// TIA Portal project "hmi_deneme" (V18)

(* hardware
DEVICE "HMI_1"  TP700 Comfort
   slot 0: "HMI_1"  TP700 Comfort  6AV2 124-0GC01-0AX0  17.0.0.0
   slot 1: "HMI_RT_1"  TP700 Comfort  6AV2 124-0GC01-0AX0  17.0.0.0
   slot 5: "HMI_1.IE_CP_1"  PROFINET Interface  17.0.0.0
      slot 1: "PROFINET Interface_1"  PROFINET Interface
         slot 1: "Port_1"  Port
         slot 2: "Port_2"  Port
   slot 7: "HMI_1.MPI/DP_CP_1"  MPI/DP Interface  17.0.0.0
DEVICE "S7-1200 station_1"  S7-1200 Station
   slot 0: "Rack_0"  S7-1200 Rack  Rack  V1.0
   slot 1: "PLC_1"  CPU 1215C DC/DC/DC  6ES7 215-1AG40-0XB0  V4.5
*)

// ===== PLC "PLC_1"  CPU 1215C DC/DC/DC =====

VAR_GLOBAL   // PLC tag table "Default tag table"
   "B0" AT %M0.0 : Bool;
   "B1" AT %M0.1 : Bool;
   "B2" AT %M0.2 : Bool;
   "B3" AT %M0.3 : Bool;
   "BTN" AT %I0.0 : Bool;
   "M0" AT %M1.0 : Bool;
   "A1" AT %M2.0 : Bool;
   "A2" AT %M2.1 : Bool;
   "M1" AT %M1.1 : Bool;
   "A3" AT %M2.2 : Bool;
   "M2" AT %M1.2 : Bool;
   "L1" AT %Q0.0 : Bool;
   "L2" AT %Q0.1 : Bool;
   "L3" AT %Q0.2 : Bool;
   "L4" AT %Q0.3 : Bool;
END_VAR

FUNCTION "Block_1" : Void   // FC1, LAD
{ S7_Optimized_Access := 'TRUE' }
VERSION : 0.1
   VAR_TEMP   // added for the SCL form of the ladder/FBD networks
      _w1 : Bool;
   END_VAR
BEGIN

REGION Network 1
   // BIT0
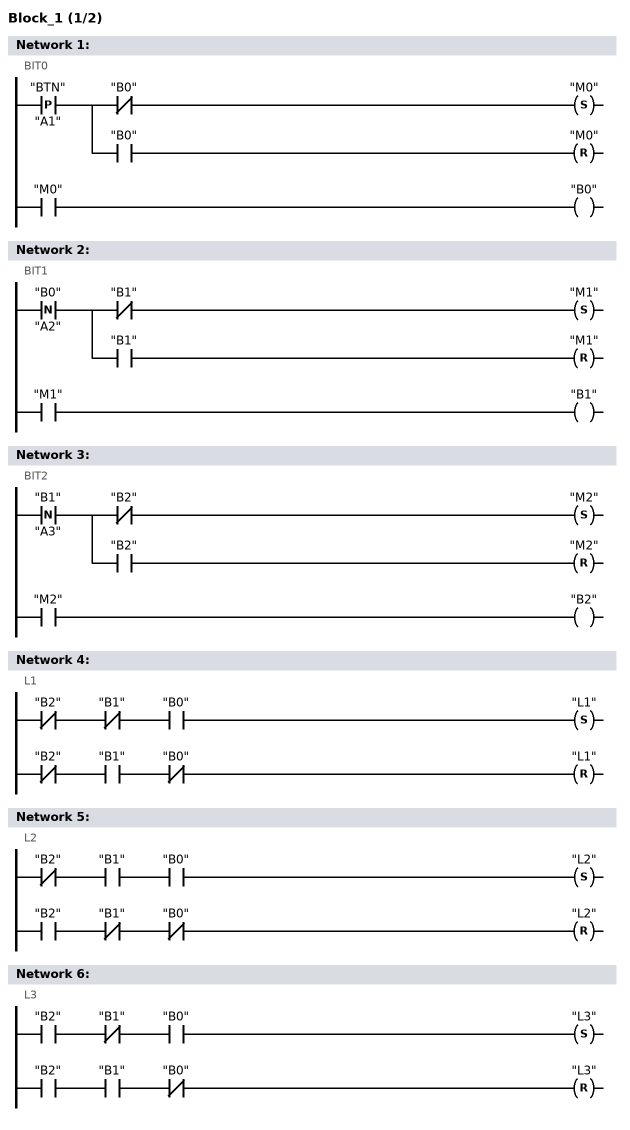
   RUNG wire#powerrail
      P_Contact(operand := "BTN", bit := "A1")
      wire#w1
      I_Contact( "B0" )
      S_Coil( "M0" )
   END_RUNG
   RUNG wire#w1
      Contact( "B0" )
      R_Coil( "M0" )
   END_RUNG
   RUNG wire#powerrail
      Contact( "M0" )
      Coil( "B0" )
   END_RUNG
   // the same network as SCL:
   #_w1 := "BTN" AND NOT "A1";   // rising edge of "BTN"
   "A1" := "BTN";
   IF #_w1 AND NOT "B0" THEN "M0" := TRUE; END_IF;
   IF #_w1 AND "B0" THEN "M0" := FALSE; END_IF;
   "B0" := "M0";
END_REGION

REGION Network 2
   // BIT1
   RUNG wire#powerrail
      N_Contact(operand := "B0", bit := "A2")
      wire#w1
      I_Contact( "B1" )
      S_Coil( "M1" )
   END_RUNG
   RUNG wire#w1
      Contact( "B1" )
      R_Coil( "M1" )
   END_RUNG
   RUNG wire#powerrail
      Contact( "M1" )
      Coil( "B1" )
   END_RUNG
   // the same network as SCL:
   #_w1 := NOT "B0" AND "A2";   // falling edge of "B0"
   "A2" := "B0";
   IF #_w1 AND NOT "B1" THEN "M1" := TRUE; END_IF;
   IF #_w1 AND "B1" THEN "M1" := FALSE; END_IF;
   "B1" := "M1";
END_REGION

REGION Network 3
   // BIT2
   RUNG wire#powerrail
      N_Contact(operand := "B1", bit := "A3")
      wire#w1
      I_Contact( "B2" )
      S_Coil( "M2" )
   END_RUNG
   RUNG wire#w1
      Contact( "B2" )
      R_Coil( "M2" )
   END_RUNG
   RUNG wire#powerrail
      Contact( "M2" )
      Coil( "B2" )
   END_RUNG
   // the same network as SCL:
   #_w1 := NOT "B1" AND "A3";   // falling edge of "B1"
   "A3" := "B1";
   IF #_w1 AND NOT "B2" THEN "M2" := TRUE; END_IF;
   IF #_w1 AND "B2" THEN "M2" := FALSE; END_IF;
   "B2" := "M2";
END_REGION

REGION Network 4
   // L1
   RUNG wire#powerrail
      I_Contact( "B2" )
      I_Contact( "B1" )
      Contact( "B0" )
      S_Coil( "L1" )
   END_RUNG
   RUNG wire#powerrail
      I_Contact( "B2" )
      Contact( "B1" )
      I_Contact( "B0" )
      R_Coil( "L1" )
   END_RUNG
   // the same network as SCL:
   IF NOT "B2" AND NOT "B1" AND "B0" THEN "L1" := TRUE; END_IF;
   IF NOT "B2" AND "B1" AND NOT "B0" THEN "L1" := FALSE; END_IF;
END_REGION

REGION Network 5
   // L2
   RUNG wire#powerrail
      I_Contact( "B2" )
      Contact( "B1" )
      Contact( "B0" )
      S_Coil( "L2" )
   END_RUNG
   RUNG wire#powerrail
      Contact( "B2" )
      I_Contact( "B1" )
      I_Contact( "B0" )
      R_Coil( "L2" )
   END_RUNG
   // the same network as SCL:
   IF NOT "B2" AND "B1" AND "B0" THEN "L2" := TRUE; END_IF;
   IF "B2" AND NOT "B1" AND NOT "B0" THEN "L2" := FALSE; END_IF;
END_REGION

REGION Network 6
   // L3
   RUNG wire#powerrail
      Contact( "B2" )
      I_Contact( "B1" )
      Contact( "B0" )
      S_Coil( "L3" )
   END_RUNG
   RUNG wire#powerrail
      Contact( "B2" )
      Contact( "B1" )
      I_Contact( "B0" )
      R_Coil( "L3" )
   END_RUNG
   // the same network as SCL:
   IF "B2" AND NOT "B1" AND "B0" THEN "L3" := TRUE; END_IF;
   IF "B2" AND "B1" AND NOT "B0" THEN "L3" := FALSE; END_IF;
END_REGION

REGION Network 7
   // L4
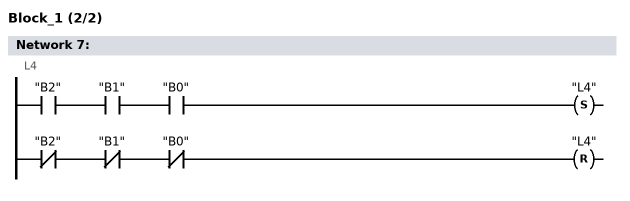
   RUNG wire#powerrail
      Contact( "B2" )
      Contact( "B1" )
      Contact( "B0" )
      S_Coil( "L4" )
   END_RUNG
   RUNG wire#powerrail
      I_Contact( "B2" )
      I_Contact( "B1" )
      I_Contact( "B0" )
      R_Coil( "L4" )
   END_RUNG
   // the same network as SCL:
   IF "B2" AND "B1" AND "B0" THEN "L4" := TRUE; END_IF;
   IF NOT "B2" AND NOT "B1" AND NOT "B0" THEN "L4" := FALSE; END_IF;
END_REGION
END_FUNCTION

ORGANIZATION_BLOCK "Main"   // OB1, LAD, ProgramCycle
TITLE = "Main Program Sweep (Cycle)"
{ S7_Optimized_Access := 'TRUE' }
VERSION : 0.1
   VAR_INPUT
      Initial_Call : Bool;   // Initial call of this OB
      Remanence : Bool;   // =True, if remanent data are available
   END_VAR
BEGIN

REGION Network 1
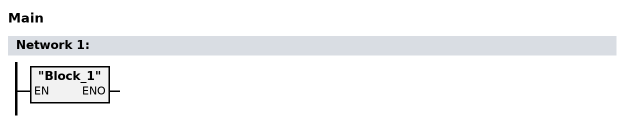
   RUNG wire#powerrail
      "Block_1"()
   END_RUNG
   // the same network as SCL:
   "Block_1"();
END_REGION
END_ORGANIZATION_BLOCK

(* ===== HMI "HMI_RT_1" =====
system functions are stored by id; their names below are inferred from use
connection "HMI_Connection_1": ETHERNET, S7_1200_OMS

HMI tags "Default tag table"
   "HMI" : Bool = PLC BTN AT %I0.0, 1 s

HMI tags "DEmo Tags"
   "Bit_1" : Bool, internal
   "Bit_2" : Bool, internal
   "Word_1" : Int, internal
   "Word_2" : Int, internal
   "AlarmTriggerWord" : UInt, internal
   "CurrentUserName" : WString[254], internal
   "CurrentGroup" : Int, internal

discrete alarms
   4: 'Warning 2', class Warnings, trigger "AlarmTriggerWord" bit 3
   3: 'Warning 1', class Warnings, trigger "AlarmTriggerWord" bit 2
   2: 'Alarm 2', class Errors, trigger "AlarmTriggerWord" bit 1
   1: 'Alarm 1', class Errors, trigger "AlarmTriggerWord" bit 0

text list "OFF_ON_List": 0 'OFF'; 1 'ON'

recipe "Recipe_1": Recipe_element_1 <- "Word_1", Recipe_element_2 <- "Word_2"

SlideinScreen "GraphX_Slidein_Left" 270x480
   TextField "Text field_1" at 28,20 size 224x23; Text 'Slide in from left screen'
   Button "Button_1" at 16,433 size 239x32; TextOff 'Close'
      on Press: function_cf6f4242("GraphX_Slidein_Left", 0)

Template "ScrNav" 800x430
   Button "Template_Button_1" at 6,391 size 192x32; TextOff 'Home'
      on Click: ActivateScreen("Home", 0)
   Button "Template_Button_2" at 205,391 size 192x32; TextOff 'Toolbox'
      on Click: ActivateScreen("Toolbox", 0)
   Button "Template_Button_3" at 404,391 size 192x32; TextOff 'Alarms'
      on Click: ActivateScreen("Alarms", 0)
   Button "Template_Button_4" at 602,391 size 192x32; TextOff 'Trend'
      on Click: ActivateScreen("Trend", 0)
   Button "Template_Button_5" at 6,353 size 192x32; TextOff 'Recipe'
      on Click: ActivateScreen("Recipe", 0)
   Button "Template_Button_6" at 205,353 size 192x32; TextOff 'UserAdmin'
      on Click: ActivateScreen("UserAdmin", 0)

screen "Home" 800x430, template "ScrNav"
   TextField "Text field_1" at 638,22 size 123x23; Text 'Home Screen'
   Button "Button_1" at 26,26 size 192x32; TextOff 'Help Popup'
      on Click: function_efd93a16("Help Popup", 0, 0, -1, -1, 1)
   Button "Button_2" at 26,73 size 192x32; TextOn 'Help Popup'; TextOff 'Show Slide in Left'
      on Press: function_cf6f4242("GraphX_Slidein_Left", 1)

screen "Toolbox" 800x430, template "ScrNav"
   TextField "Text field_1" at 629,22 size 145x23; Text 'Toolbox Screen'
   Button "Button_1" at 42,32 size 186x89; TextOff 'Momentary'; TextList "OFF_ON_List"
      on Press: function_b14e0dd5("Bit_1", 0)
      Appearance <- "Bit_1"
      ProcessValue <- "Bit_1"
   IOField "I/O field_1" at 273,32 size 93x89; FormatPattern 1
      ProcessValue <- "Bit_1"
   Circle "Circle_1" at 402,49 size 48x48
      Visibility <- "Bit_1"
   SymbolicIOField "Symbolic I/O field_1" at 480,50 size 112x46; TextOff '0'; TextOn '1'; TextList "OFF_ON_List"
      ProcessValue <- "Bit_1"

PopupScreen "Help Popup" 240x240
   Button "Button_1" at 18,198 size 197x31; TextOff 'Close'
      on Press: function_efd93a16("Help Popup", 0, 0, 0, -1, 1)
   TextField "Text field_1" at 61,34 size 108x23; Text 'Help Popup'

screen "Trend" 800x430, template "ScrNav"
   IOField "I/O field_1" at 135,14 size 96x32; FormatPattern s99999
      ProcessValue <- "Word_1"
   IOField "I/O field_2" at 395,16 size 96x32; FormatPattern s99999
      ProcessValue <- "Word_2"
   TextField "Text field_1" at 53,19 size 74x23; Text 'Word_1'
   TextField "Text field_2" at 311,19 size 74x23; Text 'Word_2'
   TrendView "Trend view_1" at 20,62 size 762x312

screen "Alarms" 800x430, template "ScrNav"
   TextField "Text field_1" at 47,38 size 226x23; Text 'Alarm Trigger Word Bits'
   IOField "I/O field_1" at 281,33 size 96x32; FormatPattern 1111
      ProcessValue <- "AlarmTriggerWord"
   AlarmView "Alarm view_1" at 49,73 size 715x165
   AlarmView "Alarm view_2" at 49,241 size 716x139

screen "Recipe" 800x430, template "ScrNav"
   IOField "I/O field_1" at 135,14 size 96x32; FormatPattern s99999
      ProcessValue <- "Word_1"
   IOField "I/O field_2" at 395,16 size 96x32; FormatPattern s99999
      ProcessValue <- "Word_2"
   TextField "Text field_1" at 53,19 size 74x23; Text 'Word_1'
   TextField "Text field_2" at 311,19 size 74x23; Text 'Word_2'
   RecipeView "Recipe view_1" at 21,57 size 753x299

screen "UserAdmin" 800x430, template "ScrNav"
   TextField "Text field_1" at 8,8 size 74x23; Text 'Word_1'
   IOField "I/O field_1" at 88,4 size 96x32; Authorization "Operate"; FormatPattern s99999
   TextField "Text field_2" at 252,13 size 185x23; Text 'Current User Name:'
   TextField "Text field_3" at 252,59 size 171x23; Text 'Current Group No:'
   TextField "Text field_4" at 629,8 size 170x23; Text 'UserAdmin Screen'
   Button "Button_1" at 692,44 size 95x49; TextOff 'Login'
      on Press: function_a2a04561()
   Button "Button_2" at 692,110 size 95x49; TextOff 'Logoff'
      on Press: function_f23ef4c9()
   Button "Button_3" at 691,206 size 96x32; TextOff 'Clear Msgs'
   IOField "I/O field_2" at 423,8 size 96x32; FormatPattern ????????????????????????????????????????????????????????????????????????????????
      ProcessValue <- "CurrentUserName"
   IOField "I/O field_3" at 422,59 size 96x32; FormatPattern s99999
      ProcessValue <- "CurrentGroup"
   AlarmView "Alarm view_1" at 30,207 size 631x131
   UserView "User view_1" at 30,106 size 481x99

VB script "VBFunction_1"
   'Tip:
   ' 1. Use the <CTRL+SPACE> or <CTRL+I> shortcut to open a list of all objects and functions
   ' 2. Write the code using the HMI Runtime object.
   '  Example: HmiRuntime.Screens("Screen_1").
   ' 3. Use the <CTRL+J> shortcut to create an object reference.
   'Write the code as of this position:

scheduled task "ChnUserTask"
   on Action: function_f41c6f6c("CurrentUserName"); function_e1ab61de("CurrentGroup"); function_de9337da()
*)